TYPE ST_PropValveMKS253:
STRUCT
	
	(* Prop valve structure, open is considered to be the higher axis position *)
	(* Note: The wiring (if using the dongle from the ALI schematic is such that the 
	stepper driver must be inverted to make the increasing counter value correspond to a more open valve. *)
	stAxis	:	AXIS_REF;
	i_HLS	AT %I*	:	BOOL; //Open
	i_LLS	AT %I*	:	BOOL; // Closed

END_STRUCT
END_TYPE

(* stored: Version 1.1.0.1, ProductVersion 3.1.4020.12
   DUT ST_PropValveMKS253: Id {73adc046-3cee-44d4-b7f7-e0e8dc3c838f} *)
